// TwinCAT 3 PLC project PLC
// ProgramVersion: 3.1.4024.0
// libraries:
//   Tc2_Standard, * (Beckhoff Automation GmbH)
//   Tc2_System, * (Beckhoff Automation GmbH)
//   Tc3_Module, * (Beckhoff Automation GmbH)
// project tree:
//   / PlcTask.TcTTO
//   POUs/ MAIN.TcPOU
// real-time tasks:
//   TASK PlcTask: cycle T#10ms, priority 20, ADS port 350

CONFIGURATION PLC
    RESOURCE PLC ON TwinCAT3
        TASK PlcTask(INTERVAL := T#10ms, PRIORITY := 20);
        PROGRAM MAIN WITH PlcTask : MAIN;
    END_RESOURCE
END_CONFIGURATION

// ---- POUs/MAIN.TcPOU
PROGRAM MAIN
VAR
	StartButton: BOOL;
	LineRun: BOOL;
	StopButton: BOOL;
	BoxConveyorRun: BOOL;
	AppleConveyorRun: BOOL;
	ctuParts: CTU;
	ApplePresent: BOOL;
	BoxPresent: BOOL;
END_VAR

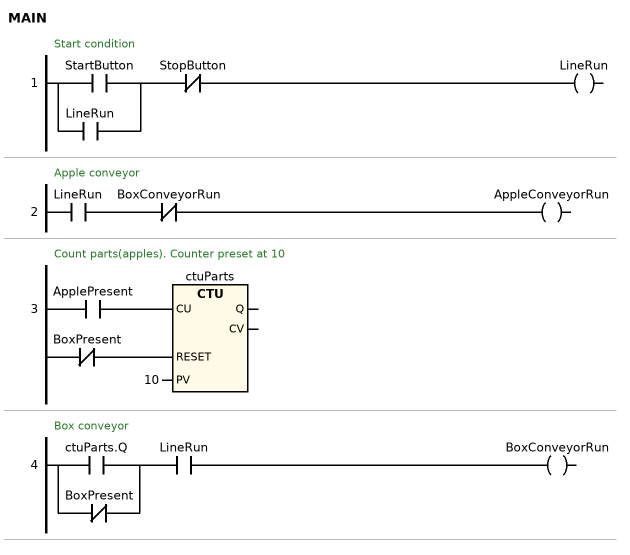
// NETWORK 1
// Start condition
LineRun := (StartButton OR LineRun) AND NOT StopButton;

// NETWORK 2
// Apple conveyor
AppleConveyorRun := LineRun AND NOT BoxConveyorRun;

// NETWORK 3
// Count parts(apples). Counter preset at 10
ctuParts(CU := ApplePresent, RESET := NOT BoxPresent, PV := 10); // CTU

// NETWORK 4
// Box conveyor
BoxConveyorRun := (ctuParts.Q OR NOT BoxPresent) AND LineRun;

END_PROGRAM
